{attribute 'linkalways'} 
{attribute 'no_explicit_call' := 'This FB is a CLASS and must be accessed using methods or properties'}
{attribute 'enable_dynamic_creation'}
FUNCTION_BLOCK _ETcVnContourApproximationMethod EXTENDS EnumDatatypeBase
VAR
	localData : ETcVnContourApproximationMethod;
	activeData : REFERENCE TO ETcVnContourApproximationMethod;
	enumBaseDatatype : _DINT(localData);
END_VAR

METHOD PRIVATE AddLocalEnumeration
VAR_INPUT
	Enumeration : T_MAXSTRING;
	Value : ETcVnContourApproximationMethod;
END_VAR
AddEnumeration(Enumeration, Value);
END_METHOD

PROPERTY PUBLIC Address : PVOID
GET
Address := ADR(activeData);
END_GET
END_PROPERTY

METHOD PUBLIC ClearReference
VAR_INPUT
END_VAR
activeData REF= localData;
SetBaseDatatypeReference();
END_METHOD

METHOD PUBLIC Clone : I_Datatype
VAR
    pClone : POINTER TO _ETcVnContourApproximationMethod;
END_VAR
pClone := __NEW(_ETcVnContourApproximationMethod(InitialValue := Value));
Clone := pClone^;
END_METHOD

METHOD FB_init : BOOL
VAR_INPUT
	bInitRetains : BOOL; // if TRUE, the retain variables are initialized (warm start / cold start)
	bInCopyCode : BOOL;  // if TRUE, the instance afterwards gets moved into the copy code (online change)
	InitialValue : ETcVnContourApproximationMethod;
END_VAR
localData := InitialValue;
AddBaseDatatype(enumBaseDatatype);
ClearReference();

AddLocalEnumeration('TCVN_CAM_NONE', ETcVnContourApproximationMethod.TCVN_CAM_NONE);
AddLocalEnumeration('TCVN_CAM_SIMPLE', ETcVnContourApproximationMethod.TCVN_CAM_SIMPLE);
AddLocalEnumeration('TCVN_CAM_TC89_L1', ETcVnContourApproximationMethod.TCVN_CAM_TC89_L1);
AddLocalEnumeration('TCVN_CAM_TC89_KCOS', ETcVnContourApproximationMethod.TCVN_CAM_TC89_KCOS);
END_METHOD

PROPERTY PUBLIC Identifier : T_MAXSTRING
GET
Identifier := 'ETcVnContourApproximationMethod';
END_GET
END_PROPERTY

METHOD IsEnumeratorValueEqual : BOOL
VAR_INPUT
	Enumerator : I_KeyValueForwardEnumerator;
END_VAR
VAR
	storedValue : ETcVnContourApproximationMethod;
END_VAR
IF NOT Enumerator.TryGet(storedValue) THEN
	RETURN;
END_IF

IsEnumeratorValueEqual := storedValue = activeData;
END_METHOD

METHOD PUBLIC MakeReferenceTo
VAR_INPUT
	ReferenceTarget : REFERENCE TO ETcVnContourApproximationMethod;
END_VAR
activeData REF= ReferenceTarget;
SetBaseDatatypeReference();
END_METHOD

METHOD PROTECTED SetBaseDatatypeReference
VAR_INPUT
END_VAR
enumBaseDatatype.MakeReferenceTo(activeData);
END_METHOD

PROPERTY PUBLIC Size : UDINT
GET
Size := SIZEOF(activeData);
END_GET
END_PROPERTY

METHOD TryMakeReferenceTo : BOOL
VAR_INPUT
	Target : I_Datatype;
END_VAR
VAR
	targetAsEnum : I_EnumDatatype;
	pTargetData : POINTER TO ETcVnContourApproximationMethod;
END_VAR
IF NOT Target.TryResolveAsEnumDatatype(targetAsEnum) THEN
	RETURN;
END_IF

IF targetAsEnum.Identifier <> Identifier THEN
	RETURN;
END_IF

pTargetData := Target.Address;
activeData REF= pTargetData^;
SetBaseDatatypeReference();
TryMakeReferenceTo := TRUE;
END_METHOD

PROPERTY PUBLIC Value : ETcVnContourApproximationMethod
GET
Value := activeData;
END_GET
SET
activeData := Value;
END_SET
END_PROPERTY

END_FUNCTION_BLOCK

(* stored: Version 1.1.0.1
   POU _ETcVnContourApproximationMethod: Id {bb3c2288-7730-4e06-857d-298d901b7641}, SpecialFunc None
   Folder Constructor: Id {5ec9adf7-0191-472b-8740-602163352476}
   Folder Private: Id {da7cb204-ed7f-4ee2-b73f-107f26ed8b7d}
   Folder Protected: Id {659b7200-c464-4520-97de-d8e32a991cfd}
   Method AddLocalEnumeration: Id {fe37461c-96df-46fa-bd38-48c727d820ec}
   Property Address: Id {98a03dc2-d80a-4961-adb4-885c59fd28d7}
   Get Get: Id {ae4c6c55-9985-4193-99a8-6fcd7d952510}
   Method ClearReference: Id {0e0c8e29-bbc8-41ec-8339-0d801a23e1ec}
   Method Clone: Id {5c5393d4-d791-4db9-a5da-4ed9966b62e1}
   Method FB_init: Id {d19dc540-a119-437a-8083-7fd40b9fa41f}
   Property Identifier: Id {b6459e86-fecc-4463-be18-ae2cd2fa9b52}
   Get Get: Id {35e16431-c352-4985-81a1-249c85e8d6a4}
   Method IsEnumeratorValueEqual: Id {53f179d6-4fbc-4b6b-804c-3e5ba4b5bbf8}
   Method MakeReferenceTo: Id {6690d58f-bb3c-4475-8a7c-8875f1adb7b3}
   Method SetBaseDatatypeReference: Id {e541f6fc-d8f8-4e4b-8893-37bf6d7f7d4c}
   Property Size: Id {f0d10ff0-6640-477e-b922-15461d3ed683}
   Get Get: Id {8dbc5dda-b1dc-465e-aeee-1ec0e08afbab}
   Method TryMakeReferenceTo: Id {db56318f-18a4-4652-b23a-6304a2caf455}
   Property Value: Id {43516786-02c0-4a8e-8647-8ba31f373492}
   Get Get: Id {459ec882-2273-4472-a444-fa9c612719ca}
   Set Set: Id {fd8bddec-325a-44af-b9f2-3a16138cb732} *)
